// TIA Portal project "time" (V14)

(* hardware
DEVICE "S7-1200 station_1"  S7-1200 Station
   slot 0: "Rack_0"  S7-1200 Rack  Rack  V1.0
   slot 1: "PLC_1"  CPU 1212C DC/DC/DC  6ES7 212-1AE40-0XB0  V4.2
*)

// ===== PLC "PLC_1"  CPU 1212C DC/DC/DC =====

VAR_GLOBAL   // PLC tag table "Default tag table"
   "start1" AT %I0.0 : Bool;
   "stop1" AT %I0.1 : Bool;
   "Tag_3" AT %I0.2 : Bool;
   "Tag_4" AT %I0.3 : Bool;
   "motor1" AT %Q0.0 : Bool;
   "motor2" AT %Q0.1 : Bool;
END_VAR

// folder: System blocks/Program resources

DATA_BLOCK "t1"   // DB1
{ S7_Optimized_Access := 'TRUE' }
AUTHOR : Simatic
FAMILY : IEC
NAME : IEC_TMR
VERSION : 1.0
// stored: InstanceOfName IEC_TIMER
"IEC_TIMER"
BEGIN
END_DATA_BLOCK

DATA_BLOCK "t2"   // DB2
{ S7_Optimized_Access := 'TRUE' }
AUTHOR : Simatic
FAMILY : IEC
NAME : IEC_TMR
VERSION : 1.0
// stored: InstanceOfName IEC_TIMER
"IEC_TIMER"
BEGIN
END_DATA_BLOCK

// folder: (top level)

ORGANIZATION_BLOCK "Main"   // OB1, LAD, ProgramCycle
TITLE = "Main Program Sweep (Cycle)"
{ S7_Optimized_Access := 'TRUE' }
VERSION : 0.1
   VAR_INPUT
      Initial_Call : Bool;   // Initial call of this OB
      Remanence : Bool;   // =True, if remanent data are available
   END_VAR
BEGIN

REGION Network 1
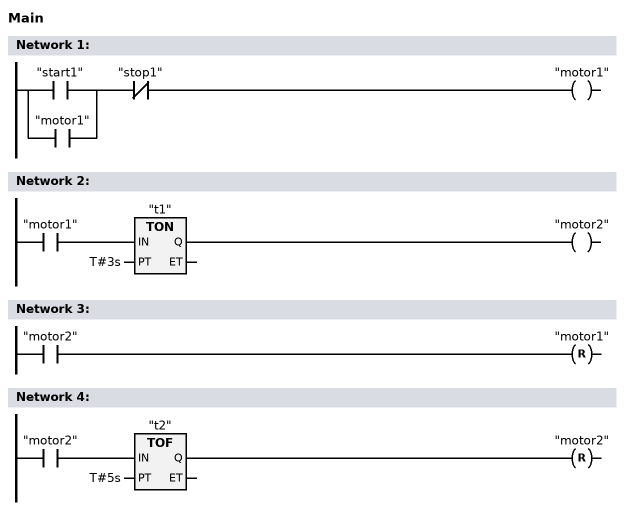
   RUNG wire#powerrail
      Contact( "start1" )
      wire#w1
      I_Contact( "stop1" )
      Coil( "motor1" )
   END_RUNG
   RUNG wire#powerrail
      Contact( "motor1" )
   END_RUNG wire#w1
   // the same network as SCL:
   "motor1" := ("start1" OR "motor1") AND NOT "stop1";
END_REGION

REGION Network 2
   "t1".TON(IN := "motor1", PT := T#3s);
   "motor2" := "t1".Q;
END_REGION

REGION Network 3
   RUNG wire#powerrail
      Contact( "motor2" )
      R_Coil( "motor1" )
   END_RUNG
   // the same network as SCL:
   IF "motor2" THEN "motor1" := FALSE; END_IF;
END_REGION

REGION Network 4
   "t2".TOF(IN := "motor2", PT := T#5s);
   IF "t2".Q THEN "motor2" := FALSE; END_IF;
END_REGION
END_ORGANIZATION_BLOCK